PROGRAM MAIN
VAR
END_VAR

END_PROGRAM

(* stored: Version 1.1.0.1
   POU MAIN: Id {8efa8018-dfe7-4c77-b084-98835f427831} *)
